TYPE ABB_STATUS_RUNNING_MODE :
(
	ABB_STATUS_RUN_UNDEF:=0, 			(* Undefined running mode *)
	ABB_STATUS_RUN_CONT_CYCLE:=1, 		(* Continuous or cycle running mode *)
	ABB_STATUS_RUN_INSTR_FWD:=2,		(* Instruction forward running mode *)
	ABB_STATUS_RUN_INSTR_BWD:=3, 		(* Instruction backward running mode *)
	ABB_STATUS_RUN_SIM:=4, 				(* Simulated running mode *)
	ABB_STATUS_RUN_STEP_MOVE:=5 		(* MOVE instructions in forward running mode and logical instructions in continuous running mode *)
);
END_TYPE

(* stored: Version 1.1.0.1, ProductVersion 3.1.4022.12
   EnumerationTextList ABB_STATUS_RUNNING_MODE: Id {601cfed0-0168-4246-86a2-501192adc3f9} *)
